FUNCTION_BLOCK FB_Convert_10V2relHum
VAR_INPUT
	iInput			:	INT;
	tRefresh		:	TIME;
END_VAR
VAR_OUTPUT
	wOut			:	WORD;
END_VAR
VAR
	rX				:	REAL;
	tonBlock		:	TON;
END_VAR

// For Convertion of 0-10V Signal from 0-100%
tonBlock(IN := NOT tonBlock.Q, PT := tRefresh);

IF tonBlock.Q THEN

	rX := iInput * 0.00030518509476; //Annahme 10V entspr. 32767
	wOut := REAL_TO_WORD(rX * 10);
	
END_IF

END_FUNCTION_BLOCK

(* stored: Version 1.1.0.1, ProductVersion 3.1.4024.4
   POU FB_Convert_10V2relHum: Id {09ca58d7-071b-400b-9162-2dfde3cf3a0a}, SpecialFunc None *)
